FUNCTION_BLOCK COLOR_DETECTOR (* Composite Function Block Type *)
  (* Standard: 61499-2 *)
  (* Version 0.0, 5/4/2023, Dmitrii, Flexbridge AB, template *)
  PACKAGE UAO.Hackathon;
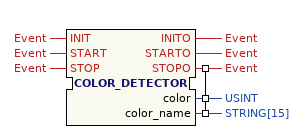
  EVENT_INPUT
    INIT; (* Initialization Request *)
    START; (* Start color detection *)
    STOP; (* Stop color detection and capture measured value. *)
  END_EVENT
  EVENT_OUTPUT
    INITO; (* Initialization Confirm *)
    STARTO; (* Color detection started *)
    STOPO WITH color, color_name; (* Color detection stopped *)
  END_EVENT
  VAR_OUTPUT
    color : USINT; (* Color code: 0='white', 1='red', 2='blue' *)
    color_name : STRING[15]; (* Color: white, red or blue *)
  END_VAR
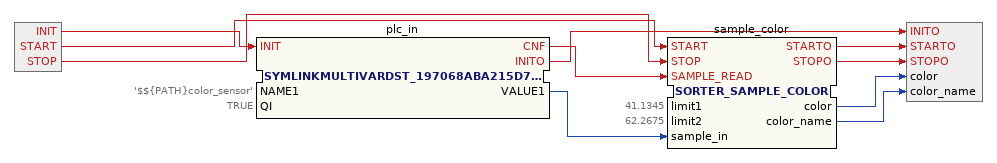
  (* NOTE: Color sensor limit values WHITE |  RED  | BLUE ^       ^ |       | limit1  limit2 *)
  FBS
    sample_color : SORTER_SAMPLE_COLOR(limit1 := 41.1345, limit2 := 62.2675);
    plc_in : SYMLINKMULTIVARDST_197068ABA215D7EBA(NAME1 := '$${PATH}color_sensor', QI := TRUE); {SET_ATTRIBUTE(Configuration.GenericFBType.InterfaceParams, Runtime.System#I:=1;VALUE${I$}:REAL)}
  END_FBS
  EVENT_CONNECTIONS
    plc_in.CNF TO sample_color.SAMPLE_READ;
    START TO sample_color.START;
    STOP TO sample_color.STOP;
    sample_color.STARTO TO STARTO;
    sample_color.STOPO TO STOPO;
    INIT TO plc_in.INIT;
    plc_in.INITO TO INITO;
  END_CONNECTIONS
  DATA_CONNECTIONS
    plc_in.VALUE1 TO sample_color.sample_in;
    sample_color.color TO color;
    sample_color.color_name TO color_name;
  END_CONNECTIONS
END_FUNCTION_BLOCK
